{attribute 'Tc2GvlVarNames'}
VAR_GLOBAL
	Presseur_Amont_K11,
	Presseur_Aval_L12	:Str_Presseur_Laser;                                          	
END_VAR

(* stored: Version 1.1.0.1, ProductVersion 3.1.4024.15
   GVL IO_PRESSEURS_LASER: Id {2215805c-02e7-42aa-b3c9-fb182b89960a} *)
